VAR_GLOBAL CONSTANT
    gcMaxPfeifferPumps	:	INT := 20; //maximum size of the Pfeiffer turbo pump array for a single port
END_VAR

(* stored: Version 1.1.0.1
   GVL GVL_PfeifferParameters: Id {7ae349b1-f7bb-4dc5-88f6-6016367034c2} *)
